{attribute 'linkalways'} 
{attribute 'no_explicit_call' := 'This FB is a CLASS and must be accessed using methods or properties'}
{attribute 'enable_dynamic_creation'}
FUNCTION_BLOCK _ETcVnEdgeDirection EXTENDS EnumDatatypeBase
VAR
	localData : ETcVnEdgeDirection;
	activeData : REFERENCE TO ETcVnEdgeDirection;
	enumBaseDatatype : _DINT(localData);
END_VAR

METHOD PRIVATE AddLocalEnumeration
VAR_INPUT
	Enumeration : T_MAXSTRING;
	Value : ETcVnEdgeDirection;
END_VAR
AddEnumeration(Enumeration, Value);
END_METHOD

PROPERTY PUBLIC Address : PVOID
GET
Address := ADR(activeData);
END_GET
END_PROPERTY

METHOD PUBLIC ClearReference
VAR_INPUT
END_VAR
activeData REF= localData;
SetBaseDatatypeReference();
END_METHOD

METHOD PUBLIC Clone : I_Datatype
VAR
    pClone : POINTER TO _ETcVnEdgeDirection;
END_VAR
pClone := __NEW(_ETcVnEdgeDirection(InitialValue := Value));
Clone := pClone^;
END_METHOD

METHOD FB_init : BOOL
VAR_INPUT
	bInitRetains : BOOL; // if TRUE, the retain variables are initialized (warm start / cold start)
	bInCopyCode : BOOL;  // if TRUE, the instance afterwards gets moved into the copy code (online change)
	InitialValue : ETcVnEdgeDirection;
END_VAR
localData := InitialValue;
AddBaseDatatype(enumBaseDatatype);
ClearReference();

AddLocalEnumeration('TCVN_ED_DARK_TO_LIGHT', ETcVnEdgeDirection.TCVN_ED_DARK_TO_LIGHT);
AddLocalEnumeration('TCVN_ED_LIGHT_TO_DARK', ETcVnEdgeDirection.TCVN_ED_LIGHT_TO_DARK);
END_METHOD

PROPERTY PUBLIC Identifier : T_MAXSTRING
GET
Identifier := 'ETcVnEdgeDirection';
END_GET
END_PROPERTY

METHOD IsEnumeratorValueEqual : BOOL
VAR_INPUT
	Enumerator : I_KeyValueForwardEnumerator;
END_VAR
VAR
	storedValue : ETcVnEdgeDirection;
END_VAR
IF NOT Enumerator.TryGet(storedValue) THEN
	RETURN;
END_IF

IsEnumeratorValueEqual := storedValue = activeData;
END_METHOD

METHOD PUBLIC MakeReferenceTo
VAR_INPUT
	ReferenceTarget : REFERENCE TO ETcVnEdgeDirection;
END_VAR
activeData REF= ReferenceTarget;
SetBaseDatatypeReference();
END_METHOD

METHOD PROTECTED SetBaseDatatypeReference
VAR_INPUT
END_VAR
enumBaseDatatype.MakeReferenceTo(activeData);
END_METHOD

PROPERTY PUBLIC Size : UDINT
GET
Size := SIZEOF(activeData);
END_GET
END_PROPERTY

METHOD TryMakeReferenceTo : BOOL
VAR_INPUT
	Target : I_Datatype;
END_VAR
VAR
	targetAsEnum : I_EnumDatatype;
	pTargetData : POINTER TO ETcVnEdgeDirection;
END_VAR
IF NOT Target.TryResolveAsEnumDatatype(targetAsEnum) THEN
	RETURN;
END_IF

IF targetAsEnum.Identifier <> Identifier THEN
	RETURN;
END_IF

pTargetData := Target.Address;
activeData REF= pTargetData^;
SetBaseDatatypeReference();
TryMakeReferenceTo := TRUE;
END_METHOD

PROPERTY PUBLIC Value : ETcVnEdgeDirection
GET
Value := activeData;
END_GET
SET
activeData := Value;
END_SET
END_PROPERTY

END_FUNCTION_BLOCK

(* stored: Version 1.1.0.1
   POU _ETcVnEdgeDirection: Id {8ffa9ee8-9489-4c3c-909c-df7b59f5d60a}, SpecialFunc None
   Folder Constructor: Id {107b945e-889d-4f79-b46c-cb5f040677fd}
   Folder Private: Id {80f12c22-7c94-44f4-b3c0-66a553502e57}
   Folder Protected: Id {61e1034e-b071-482a-a01e-d7eebe638371}
   Method AddLocalEnumeration: Id {4f7f6f30-8f40-4948-bb75-90c4b4b9be90}
   Property Address: Id {881984b2-f4b0-49c1-ad57-c05e86cccafe}
   Get Get: Id {b90498a3-d217-4ccd-86c1-493881792e3d}
   Method ClearReference: Id {6e4fe68d-9e1f-49b6-bfbd-3e9ba2ed2127}
   Method Clone: Id {5d69ce10-7dda-4c66-9439-91c9e73c8fd8}
   Method FB_init: Id {a7b7f2d9-d62a-416c-abb6-b1f3c9ceea8d}
   Property Identifier: Id {53bb8755-3662-4d24-9083-6c035a69bb3c}
   Get Get: Id {ffd354fd-d09b-4ed1-9e89-2f3246880255}
   Method IsEnumeratorValueEqual: Id {efa46f25-85ef-4ff4-a0eb-02e6be6771c7}
   Method MakeReferenceTo: Id {84d762ac-b0ff-48d2-b600-5b8a7a0db69d}
   Method SetBaseDatatypeReference: Id {698ae87a-cabf-4eb9-979c-cafa3b852b63}
   Property Size: Id {6542c675-9f86-4ac4-b065-341e70db769b}
   Get Get: Id {8029b012-ceb5-43b3-af1f-da72cdcc317f}
   Method TryMakeReferenceTo: Id {c7721b44-a356-4e30-9154-5e064629c7b3}
   Property Value: Id {beec4843-ec87-4907-8468-565c0ec6de3b}
   Get Get: Id {ba48b5d9-9059-481a-b701-a3f7d9764f9b}
   Set Set: Id {e0897230-d034-4a38-8d96-2502ac81f27f} *)
